FUNCTION_BLOCK FB_MOD_INT (* IEC 61131-3,Table 24#16 *)
  (* Standard: 61131-3 *)
  (* Version 0.1, 2006-09-12, JHC, Holobloc Inc, Moved to fb.rt.math. *)
  (* Version 0.0, 2004-12-15, JHC, Rockwell Automation, Converted from SRC format. *)
  (* Compiler header: package fb.rt.math; *)
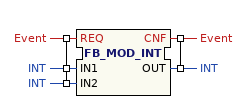
  EVENT_INPUT
    REQ WITH IN1, IN2;
  END_EVENT
  EVENT_OUTPUT
    CNF WITH OUT;
  END_EVENT
  VAR_INPUT
    IN1 : INT;
    IN2 : INT;
  END_VAR
  VAR_OUTPUT
    OUT : INT;
  END_VAR
END_FUNCTION_BLOCK
